FUNCTION_BLOCK Data_Scope_1
  (* Standard: 61499-2 *)
  (* Version 03-07-12, GASR *)
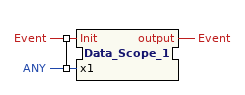
  EVENT_INPUT
    Init WITH x1;
  END_EVENT
  EVENT_OUTPUT
    output;
  END_EVENT
  VAR_INPUT
    x1 : ANY;
  END_VAR
  SERVICE Data_Scope_1/USER
    SEQUENCE seq1
      Data_Scope_1.Init() -> USER.req();
      USER.rsp() -> Data_Scope_1.output();
    END_SEQUENCE
  END_SERVICE
END_FUNCTION_BLOCK
